FUNCTION Convert_ULINT_TO_LREAL : Hresult
VAR_INPUT
	in : ULINT;
	out : REFERENCE TO LREAL;
END_VAR
VAR
	converted : LREAL;
END_VAR
VAR CONSTANT
	INCOMPATIBLE : HRESULT := 16#9811070E;
END_VAR

converted := ULINT_TO_LREAL(in);

IF (LREAL_TO_ULINT(converted) <> in) THEN
	Convert_ULINT_TO_LREAL := INCOMPATIBLE;
	RETURN;
END_IF

out := converted;

END_FUNCTION

(* stored: Version 1.1.0.1, ProductVersion 3.1.4024.12
   POU Convert_ULINT_TO_LREAL: Id {fa9ff760-4e57-4046-9057-a9980c9c9d5d}, SpecialFunc None *)
